INTERFACE ITF_Writer

METHOD WriteMessage : BOOL
VAR_INPUT
	SomeString : STRING(80);
END_VAR
END_METHOD

END_INTERFACE

(* stored: Version 1.1.0.1, ProductVersion 3.1.4024.12
   Itf ITF_Writer: Id {a64e0f6d-d113-44bb-92cb-ccd3345a0e25}
   Method WriteMessage: Id {ea160ff3-f226-4021-91d9-0644a31e4034} *)
